{attribute 'GeneratedUsingTerminal: AMP8000-0030-0103-0103'}
{attribute addProperty BoxType "AMP8000-0030-0103-0103"}
{attribute addProperty Id "FSOEAT %I*FSOE_31BB7F2A21"}
{attribute addProperty CRC "856307172"}
{attribute addProperty Size "21"}
TYPE FSoE_Slave_Connection_1_Slave_Message_330A35E4 :
STRUCT
	{attribute addProperty Name "FSOE"}
	FSOE AT %I* : FSOE_31BB7F2A;
END_STRUCT
END_TYPE

(* stored: Version 1.2.0.0, ProductVersion 3.1.4024.9
   DUT FSoE_Slave_Connection_1_Slave_Message_330A35E4: Id {42b96ad6-cc4c-4465-986e-6b11c853aebe} *)
